FUNCTION_BLOCK MC_TORQUELIMITING
VAR_INPUT
	{attribute 'hide'} 
	Axis : AXIS_REF;
	Enable : BOOL;
	TLimit : LREAL;
	Mode : DINT;
END_VAR
VAR_OUTPUT
	InClamping : BOOL;
	InLimitation : BOOL;
	Busy : BOOL;
	Error : BOOL;
	ErrorId : WORD;
END_VAR
VAR
END_VAR

;

END_FUNCTION_BLOCK

(* stored: Version 1.1.0.1
   POU MC_TORQUELIMITING: Id {8df7729b-15f5-4ef9-b84f-163c7a4b6dc7}, SpecialFunc None *)
